(* CoDeSys 2.3 export: ST_MQTTRECEIVEDPUBLISHTELEGRAM.EXP *)

(* Data type *)
TYPE ST_MqttReceivedPublishTelegram :
STRUCT
	sTopic		: STRING[255];
	sValue		: STRING[255];
	bHasData	: BOOL;
END_STRUCT
END_TYPE
